// TIA Portal V20 export
DATA_BLOCK "DB_MiscPLC_IHM_ISO"   // DB97
// stored: InstanceOfName FB_MiscPLC_IHM_ISO, InstanceOfType FB
"FB_MiscPLC_IHM_ISO"
   // VAR
   //    sTransferSelData { S7_SetPoint := 'True'} : Array[0..11] of Byte;
   //    sTransferActData : Array[0..11] of Byte;
   //    sUpdate_PLC_ISO_Values : Bool;
   //    sRT_bStopAfterEmptying : R_TRIG;
   //    sRT_CNCModeReq { S7_SetPoint := 'True'} : R_TRIG;
   // END_VAR
BEGIN
END_DATA_BLOCK
